(* PLC project motor_2dir_1speed, Dassault Systèmes ControlBuild 2024x *)
(* stored: creationDateTime 2023-10-03T11:13:09-01:00 *)

(* This module simulates the behaviour of a motor with 2 directions and 1speed and its electrical control logic. *)
FUNCTION_BLOCK equipment_library.motor_2dir_1speed
  VAR_INPUT
    voltage380 : BOOL := true;
    cmdSupply : BOOL := true;
    sensorSupply : BOOL := true;
  END_VAR
  VAR_INPUT
    forward : BOOL := false;
    backward : BOOL := false;
  END_VAR
  VAR_OUTPUT
    forwardFB : BOOL := false;
    backwardFB : BOOL := false;
    thermal : BOOL := false;
  END_VAR
  VAR_OUTPUT
    speedVal : REAL := 0.0;
    speedPercent : REAL := 0.0;
  END_VAR
  VAR
    increment : REAL := 0.0;
    memoFwd : BOOL := false;
    memoBwd : BOOL := false;
    forwardState : BOOL := false;
    backwardState : BOOL := false;
    wantedSpeed : REAL := 0.0;
  END_VAR
  VAR CONSTANT
    nominalSpeed : REAL := 5000.0;
    nominalTime : REAL := 0.5;
    thermalLogic : BOOL := false;
    fwdFbLogic : BOOL := true;
    bwdFbLogic : BOOL := true;
  END_VAR
  VAR
    d_locking : BOOL := false;
    v_d_locking : REAL := 0.0;
    d_electrical : BOOL := false;
    v_d_electrical : BOOL := false;
    d_backwardFB : BOOL := false;
    v_d_backwardFB : BOOL := false;
    d_forwardFB : BOOL := false;
    v_d_forwardFB : BOOL := false;
  END_VAR


ACTION C_source_code:
/* ----------------------------------------------------------------	*/
/* Type : Model of Operative Behaviour					*/
/* Category :  Associations - motors					*/
/* Author : Dassault Systemes						*/
/* Update date : June 2018							*/
/* ----------------------------------------------------------------	*/
/* This module simulates a motor with 2 directions and 1 speed	*/
/* and its electrical control logic.					*/
/* ----------------------------------------------------------------	*/


/* ----------------------------------------------------------------	*/
/* Management of orders from Control Part					*/
/*	if there is no power supply for command 				*/
/*     	the contactors don't understand the control order	*/
/*	The contactors cannot be active in the same time		*/
/*	 	(mechanical security).					*/
/* ----------------------------------------------------------------	*/
if (forward && !memoBwd && cmdSupply) memoFwd = 1;
if (!forward || !cmdSupply || d_electrical) memoFwd = 0;
if (!memoFwd && backward && cmdSupply) memoBwd = 1;
if (!backward || !cmdSupply || d_electrical) memoBwd = 0;

/* ----------------------------------------------------------------	*/
/* Calculation of the on-state of contactor				*/
/* ----------------------------------------------------------------	*/
forwardState= memoFwd & voltage380;
backwardState = memoBwd & voltage380;


/* ----------------------------------------------------------------	*/
/* Management of the speed ramp						*/
/* ----------------------------------------------------------------	*/
if (d_locking)  speedVal = v_d_locking;
else {
	/* Compute the increment of translation according to the simulation clock	*/
	if (nominalTime > 0.0)
		increment = (nominalSpeed / nominalTime) * (CLOCK_PERIOD/1000000.0);

	/* Compute the wanted speed	*/
	if (forwardState) wantedSpeed = nominalSpeed;
	if (backwardState) wantedSpeed = nominalSpeed * -1.0;
	if (! forwardState && ! backwardState) wantedSpeed = 0.0;

	/* Compute the speed ramp	*/
	if ( speedVal < wantedSpeed ) {
		speedVal += increment;
		if (speedVal > wantedSpeed)  speedVal = wantedSpeed;
	}
	if ( speedVal > wantedSpeed ) {
		speedVal -= increment;
		if (speedVal < wantedSpeed)  speedVal = wantedSpeed;
	}
}

/* ----------------------------------------------------------------	*/
/* Compute the percentage between the current and nominal speed	*/
/* ----------------------------------------------------------------	*/
if (nominalSpeed != 0.0) 
	speedPercent = ((speedVal/nominalSpeed)*100);


/* ----------------------------------------------------------------	*/
/* Management of the thermal feedback					*/
/* ----------------------------------------------------------------	*/
if (d_electrical) thermal=v_d_electrical;
else
	thermal= ! thermalLogic && sensorSupply;


/* ----------------------------------------------------------------	*/
/* Management of feedback to Control Part					*/
/*     if a fault is required, the contactor feed-back 		*/
/*		 takes a preset state.					*/
/*	if there is no power supply for sensors 				*/
/*         contactor feed-back returns nothing				*/
/*     else contactor feed-back returns the contactor state combined	*/
/*	    with wiring logic.						*/
/* ----------------------------------------------------------------	*/
if (d_forwardFB) forwardFB=v_d_forwardFB;
else
	forwardFB=(memoFwd ^ ! fwdFbLogic) && sensorSupply;

if (d_backwardFB) backwardFB=v_d_backwardFB;
else
	backwardFB=(memoBwd ^ ! bwdFbLogic) && sensorSupply;
END_ACTION
END_FUNCTION_BLOCK
